FUNCTION_BLOCK E_MOVE (* Data latch (d) flip flop for ANY Datatype *)
  (* Standard: 61499; Classification: Sample and Hold; Description: Copyright (c) 2013, 2024 TU Wien ACIN,  HR Agrartechnik GmbH This program and the accompanying materials are made available under the terms of the Eclipse Public License 2.0 which is available at https://www.eclipse.org/legal/epl-2.0/ SPDX-License-Identifier: EPL-2.0 This Block is functional identic to E_D_FF but for ANY Datatype. it reduces the Number of Events on the Output CNF. This Block take the input IN compare it with the output OUT and only if it is not equal forward the event REQ to CNF. for REAL and LREAL the Function of this Block is not guaranteed, because of the special cases of rounding Errors in REAL and LREAL. *)
  (* Version 1.0, 2013-08-17, Monika Wenger, TU Wien ACIN *)
  (* Version 1.1, 2024-10-31, Franz Höpfinger, HR Agrartechnik GmbH, Copy F_MOVE to E_MOVE and adjust Comments *)
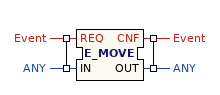
  EVENT_INPUT
    REQ WITH IN; (* Normal Execution Request *)
  END_EVENT
  EVENT_OUTPUT
    CNF WITH OUT; (* Execution Confirmation *)
  END_EVENT
  VAR_INPUT
    IN : ANY; (* input *)
  END_VAR
  VAR_OUTPUT
    OUT : ANY; (* input = output *)
  END_VAR
END_FUNCTION_BLOCK
